// TIA Portal V17 export
// export: Created 2024-09-02T12:50:36.8295845Z, ExportSetting WithDefaults, DisplayName Totally Integrated Automation Portal, DisplayVersion V17, DisplayName TIA Portal Openness, DisplayVersion V17, DisplayName TIA Portal Version Control Interface, DisplayVersion V17, DisplayName STEP 7 Professional, DisplayVersion V17, DisplayName STEP 7 Safety, DisplayVersion V17, DisplayName WinCC Professional, DisplayVersion V17
TYPE "TypeMobyDatenPuffer"
// stored: IsFailsafeCompliant false
   STRUCT
      "Byte" : Array[0..63999] of Byte;
   END_STRUCT;
END_TYPE
